TYPE sAnalogSim :
STRUCT
	simEnable : BOOL := FALSE;
	simValue : LREAL := 0.0;
END_STRUCT
END_TYPE

(* stored: Version 1.1.0.1, ProductVersion 3.1.0.36
   DUT sAnalogSim: Id {a5ed2743-07cc-440b-b482-0c8ef0cd086e} *)
